TYPE ST_ScrewdriverMotionConfig :
STRUCT
    stY : ST_VelocityConfig;
    stZ : ST_VelocityConfig;
    fPositionTolerance : LREAL;
    tMoveTimeout : TIME;
END_STRUCT
END_TYPE

(* stored: Version 1.1.0.1, ProductVersion 3.1.4026.20
   DUT ST_ScrewdriverMotionConfig: Id {6e1d9805-cd94-4c30-90b7-93bb9bb6b565} *)
